FUNCTION_BLOCK FIFO_StateTrace
VAR_INPUT
	Overwrite	: BOOL;							// Flag to Overwrite FIFO Elements (when filled)
	pFIFO		: POINTER TO TraceFIFOBuffer;	// Pointer to FIFO Memory
END_VAR

VAR_OUTPUT
	Error		: BOOL;							// Flag Indicating Error with FIFO
	Count		: DINT;							// Count of Elements Within FIFO
	Full		: BOOL;							// Flag Indicating FIFO Full
END_VAR

VAR
	Head		: UDINT;						// Index of Head Element (Newest)
	Tail		: UDINT;						// Index of Tail Element (Oldest)
END_VAR

ACTION INIT:
// Clear Buffer and Output Data
MEMSET(ADR(pFIFO^.Buffer), 0, SIZEOF(pFIFO^.Buffer));

// Reset Count / Indicies
Count 	:= 0;
Head 	:= 0;
Tail 	:= 0;

// Reset Flags
Full 	:= FALSE;
Error 	:= FALSE;
END_ACTION

METHOD LOAD : BOOL
VAR_INPUT
	Input	: StatsEvent;
END_VAR
// Set Success Flag
Error := FALSE;
LOAD := TRUE;

// Check if FIFO Has Room (or Overwrite Enabled)
IF (Full AND Overwrite) OR NOT Full THEN
	
	// Set Head Element to Input Value
	pFIFO^.Buffer[Head] := Input;
	
	// Iterate Head Index
	Head := Head + 1;
	
	// Check if Head at Maximum Value, Rollover
	IF Head = pFIFO^.Size THEN
		Head := 0;
	END_IF
	
	// If FIFO Full, Iterate Tail
	IF Full THEN
		Tail := Tail + 1;
		
		// If Tail at Maximum Value, Rollover
		IF Tail = pFIFO^.Size THEN
			Tail := 0;
		END_IF
		
	// Otherwise Update Count
	ELSE
		Count := Count + 1;
	END_IF
	
// Otherwise, Flag Failure (Value Appended to Full FIFO)
ELSE
	Error := TRUE;
	LOAD := FALSE;
	
END_IF

Full := Head = Tail;
END_METHOD

METHOD PEEK : StatsEvent
// Reset Error Flag
Error := FALSE;

// Check if FIFO Full or Tail
IF Count > 0 THEN
	PEEK := pFIFO^.Buffer[Tail];
	
// Otherwise, Flag Error (FIFO is Empty)
ELSE
	Error := TRUE;
END_IF
END_METHOD

METHOD UNLOAD : StatsEvent
// Reset Error Flag
Error := FALSE;

// Check if FIFO Has Elements
IF Count > 0 THEN
	
	// Fetch Oldest Value from FIFO
	UNLOAD := pFIFO^.Buffer[Tail];
	
	// Clear FIFO Position
	pFIFO^.Buffer[Tail] := 0; 
	
	// Update Oldest Value Index
	Tail := Tail + 1;
	
	// Update Element Count
	Count := Count - 1;
	
	// Check for Rollover
	IF Tail = pFIFO^.Size THEN
		Tail := 0;
	END_IF
	
	// Reset Full Flag
	Full := FALSE;
	
// Otherwise, Flag Error (FIFO is Empty)
ELSE
	Error 	:= TRUE;
	UNLOAD := 0;
END_IF
END_METHOD

END_FUNCTION_BLOCK

(* stored: Version 1.1.0.1, ProductVersion 3.1.4024.9
   POU FIFO_StateTrace: Id {3351118f-bba1-4382-8094-400dc0b7365c}, SpecialFunc None
   Action INIT: Id {56528050-524d-446c-8d5e-5ab96d2b6147}
   Method LOAD: Id {4295ba78-5e0c-42c0-a74f-f7b856ffb2f1}
   Method PEEK: Id {d0110137-52f1-481a-9a0b-e81ed44d63e1}
   Method UNLOAD: Id {2ce9905e-ccbe-4445-8489-2173700b7ae8} *)
